// TwinCAT 3 PLC project Aufgabenserie4
// ProgramVersion: 3.1.4022.3
// libraries:
//   Tc2_Standard, * (Beckhoff Automation GmbH)
//   Tc2_System, * (Beckhoff Automation GmbH)
//   Tc3_Module, * (Beckhoff Automation GmbH)
// project tree:
//   / GlobalTextList.TcGTLO, PlcTask.TcTTO, Visualisierungsmanager.TcVMO (not stored)
//   GVLs/ GVL.TcGVL
//   POUs/ Integrator.TcPOU, LowpassFilter.TcPOU, MAIN.TcPOU
//   VISUs/ Visualization.TcVIS
// real-time tasks:
//   TASK PlcTask: cycle T#10ms, priority 20, ADS port 350

CONFIGURATION Aufgabenserie4
    RESOURCE PLC ON TwinCAT3
        TASK PlcTask(INTERVAL := T#10ms, PRIORITY := 20);
        PROGRAM MAIN WITH PlcTask : MAIN;
    END_RESOURCE
END_CONFIGURATION

// ---- GVLs/GVL.TcGVL
{attribute 'qualified_only'}
VAR_GLOBAL
	i_TasterYellow AT%I* : BOOL;
END_VAR

// ---- POUs/MAIN.TcPOU
PROGRAM MAIN
VAR
	r_Tao : REAL := 0.1;
	r_Input : REAL;;
	r_Output : REAL;
	FB_LowPasss : LowpassFilter;
END_VAR

FB_LowPasss();
FB_LowPasss.r_Tao := r_Tao;
IF
FB_LowPasss.r_Input := r_Input;
r_Output := FB_LowPasss.r_Output;

END_PROGRAM

// ---- POUs/LowpassFilter.TcPOU
FUNCTION_BLOCK LowpassFilter
VAR_INPUT
	r_Input : REAL;
	r_Tao : REAL;
END_VAR
VAR_OUTPUT
	r_Output : REAL;
END_VAR
VAR
	r_Output_k1 : REAL;
	r_Time : REAL := 0.01;
END_VAR

r_Output := (r_Input + (r_Input*r_Tao/r_Time))/(1+r_Tao/r_Time);
r_Output_k1 := r_Output;

END_FUNCTION_BLOCK

// ---- POUs/Integrator.TcPOU
FUNCTION_BLOCK Integrator
VAR_INPUT
END_VAR
VAR_OUTPUT
END_VAR
VAR
END_VAR

END_FUNCTION_BLOCK

// ---- VISUs/Visualization.TcVIS
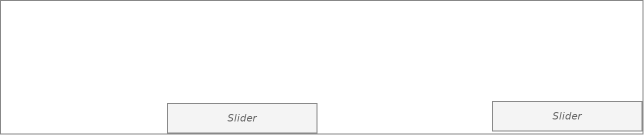
VISUALIZATION Visualization  // 644x135
    Slider (167,103 150x30), variable: MAIN.r_Tao, scale 0..10
    Slider (492,101 150x30), variable: MAIN.r_Input, scale 0..100
END_VISUALIZATION
